// TIA Portal V15 export
// export: Created 2018-05-30T13:29:09.7161607Z, ExportSetting WithDefaults, WithReadOnly, DisplayName Totally Integrated Automation Portal, DisplayVersion V15, DisplayName TIA Portal Openness, DisplayVersion V15, DisplayName STEP 7 Professional, DisplayVersion V15, DisplayName WinCC Professional, DisplayVersion V15
FUNCTION_BLOCK "BST_VALVE_400"   // FB20, STL
{ S7_Optimized_Access := 'FALSE' }
VERSION : 0.1
// stored: AutoNumber false, CodeModifiedDate 2018-05-30T13:28:59.5225777Z, CompileDate 2018-05-30T13:28:59.5215776Z, CreationDate 2018-05-30T13:22:11.3692328Z, InterfaceModifiedDate 2018-05-30T13:23:22.3522927Z, IsConsistent true, IsKnowHowProtected false, ISMultiInstanceCapable true, IsWriteProtected false, LibraryConformanceStatus The object is library-conformant., ModifiedDate 2018-05-30T13:28:59.5225777Z, ParameterModified 2018-05-30T13:23:22.3522927Z, StructureModified 2018-05-30T13:23:22.3522927Z, UDAEnableTagReadback false
   VAR_INPUT
      AUT_OP : Bool;   // Auto command from program
      FB_OPEN : Bool;   // Feedback Open
      FB_CLOSE : Bool;   // Feedback Close
   END_VAR
   VAR_OUTPUT
      QOPEN : Bool;   // Opened
      QCLOSE : Bool;   // Closed
      QMON_ERR : Bool;   // Monitoring Error
      QCMD_OP : Bool;   // Command to Valve
   END_VAR
BEGIN
END_FUNCTION_BLOCK
